Staubli VAL3: Deb2403.dtx

mdesc mNomSpeed = {accel=200, vel=400, decel=200, blend=cartesian}
tool tTool = {z=67, fatherId=flange[0], ioLink=valve1}
jointRx jP1
jointRx jP2 = {j1=67.72, j2=50.87, j3=100.24, j5=28.89, j6=-112.28}
jointRx jP3 = {j1=-83.94, j2=66.93, j3=62.59, j5=50.48, j6=-263.94}
jointRx jP4 = {j1=67.72, j2=17.89, j3=90, j5=72.11, j6=-112.28}
jointRx jP5 = {j1=-84.94, j2=43.97, j3=50.35, j5=58.68, j6=-263.94}
frame fFrame = {x=-421.67, y=-92.07, z=-232.31, rx=0.62, ry=178.2, rz=-83.18, fatherId=world[0]}
public dio diECAT1_0 = {link=POWERLINK-1\%I0}
public dio diECAT1_1 = {link=POWERLINK-1\%I1}
public dio diECAT1_2 = {link=POWERLINK-1\%I2}
public dio diECAT1_3 = {link=POWERLINK-1\%I3}
public dio diECAT1_4 = {link=POWERLINK-1\%I4}
public dio diECAT1_5 = {link=POWERLINK-1\%I5}
public dio diECAT1_6 = {link=POWERLINK-1\%I6}
public dio diECAT1_7 = {link=POWERLINK-1\%I7}
public dio diECAT1_8 = {link=POWERLINK-1\%I8}
public dio diECAT1_9 = {link=POWERLINK-1\%I9}
public dio diECAT1_10 = {link=POWERLINK-1\%I10}
public dio diECAT1_11 = {link=POWERLINK-1\%I11}
public dio diECAT1_12 = {link=POWERLINK-1\%I12}
public dio diECAT1_13 = {link=POWERLINK-1\%I13}
public dio diECAT1_14 = {link=POWERLINK-1\%I14}
public dio diECAT1_15 = {link=POWERLINK-1\%I15}
public dio diECAT1_16 = {link=POWERLINK-1\%I16}
public dio doECAT1_0 = {link=POWERLINK-1\%Q0}
public dio doECAT1_1 = {link=POWERLINK-1\%Q1}
bool rbt_ready
num co_x
num co_y
num nPowerlink
num y[8]
num x[8]
pointRx pPointRx = {x=-421.67, y=-92.07, z=-232.31, rx=0.62, ry=178.2, rz=-83.18, fatherId=world[0]}
trsf trTrsf
pointRx pPoint1[2]
  [0] = {x=86.09, y=-273.22, z=67.88, rx=179.43, ry=-0.9, rz=19.53, fatherId=world[0]}
  [1] = {x=261.8, y=34.46, z=106.21, rx=179.25, ry=0.27, rz=-60, fatherId=world[0]}
